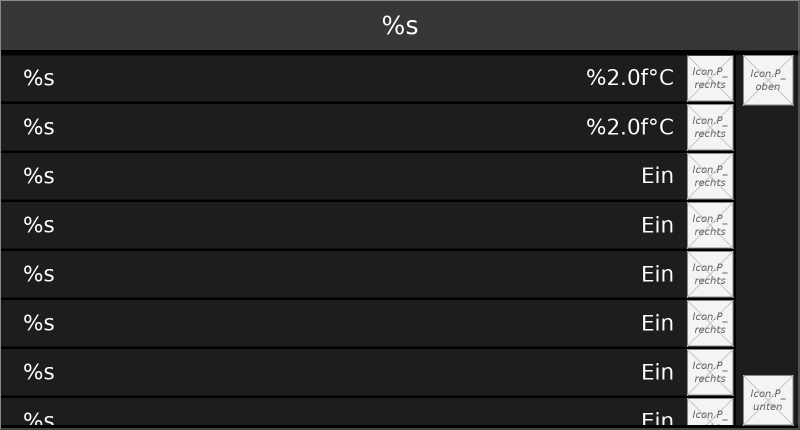
VISUALIZATION SW_WG_UWP_Verd_Liste  // 800x430
VAR_IN_OUT
	FB_GR2:GR_2;
END_VAR

VAR_INPUT
	i_Titel:INT;
END_VAR

VAR
	i_verschieben:INT;
 END_VAR
    Rectangle (0,55 733x46)
    Label (20,55 479x46), "%s"
    Rectangle (0,104 733x46)
    Label (20,104 479x46), "%s"
    Rectangle (547,55 130x45), "%2.0f°C", text variable: FB_GR2.f_AT
    Rectangle (547,104 130x46), "%2.0f°C", text variable: FB_GR2.f_RefPunkt_TO1
    Image (687,55 46x46), image: Icon.P_rechts
        OnMouseClick: execute { GWP_Library.Visu.i_Frame_Index:=1; }
    Image (687,104 46x46), image: Icon.P_rechts
    Rectangle (0,153 733x46)
    Label (20,153 479x46), "%s"
    Rectangle (0,202 733x46)
    Label (20,202 479x46), "%s"
    Rectangle (0,251 733x46)
    Label (20,251 479x46), "%s"
    Rectangle (0,300 733x46)
    Label (20,300 479x46), "%s"
    Rectangle (0,349 733x46)
    Label (20,349 479x46), "%s"
    Rectangle (0,398 733x46)
    Label (20,398 479x46), "%s"
    Rectangle (0,447 733x46)
    Label (20,447 479x46), "%s"
    Rectangle (0,496 733x46)
    Label (20,496 479x46), "%s"
    Rectangle (0,545 733x46)
    Label (20,545 479x46), "%s"
    Rectangle (547,153 130x45), "Ein"
    Rectangle (547,202 130x46), "Ein"
    Rectangle (547,251 130x46), "Ein"
    Rectangle (547,300 130x46), "Ein"
    Rectangle (547,349 130x46), "Ein"
    Rectangle (547,447 130x46), "Ein"
    Rectangle (547,398 130x46), "Ein"
    Rectangle (547,496 130x46), "Ein"
    Rectangle (547,545 130x46), "Ein"
    Image (687,153 46x46), image: Icon.P_rechts
        OnMouseClick: execute { GWP_Library.Visu.i_Frame_Index:=3; }
    Image (687,545 46x46), image: Icon.P_rechts
    Image (687,496 46x46), image: Icon.P_rechts
    Image (687,447 46x46), image: Icon.P_rechts
    Image (687,398 46x46), image: Icon.P_rechts
    Image (687,349 46x46), image: Icon.P_rechts
    Image (687,300 46x46), image: Icon.P_rechts
    Image (687,251 46x46), image: Icon.P_rechts
    Image (687,202 46x46), image: Icon.P_rechts
    Rectangle (0,594 733x46)
    Label (20,594 479x46), "%s"
    Rectangle (547,594 130x45), "Ein"
    Image (687,594 46x46), image: Icon.P_rechts
    Image (79,430 50x50), image: Icon.zurueck
        OnMouseClick:  Assign=Sollwertmenu_Waermegewinnung, Type=Assignment
        OnMouseClick: execute { i_verschieben:=0; }
    Rectangle (0,0 800x50), "%s", text list: 'Sprachen', text index: i_Titel
    Group (736,55 64x370)
        Rectangle (0,0 64x370)
        Image (7,320 50x50), image: Icon.P_unten
            OnMouseClick: execute {
                IF i_verschieben<0 THEN
                	i_verschieben:=i_verschieben+53;
                End_if
            }
        Image (7,0 50x50), image: Icon.P_oben
            OnMouseClick: execute {
                IF  i_verschieben>-200 THEN
                	i_verschieben:=i_verschieben-53;
                End_if
            }
    Rectangle (0,50 733x5)
    Rectangle (0,425 733x5)
END_VISUALIZATION

// VISUs/Sollwertmenu_9/Wärmegewinnung/Sollwertmenu_Waermegewinnung
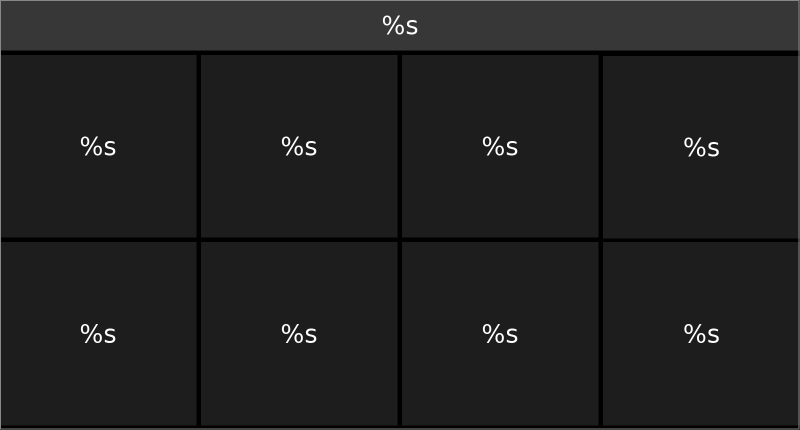
VISUALIZATION Sollwertmenu_Waermegewinnung  // 800x430
    Rectangle (0,0 800x50), "%s", text list: 'Sprachen', text index: 4
    Rectangle (0,55 196x182), "%s", text list: 'Sprachen', text index: 5
        OnMouseClick:  Assign=SW_WG_UWP_Verd, Type=Assignment
    Rectangle (201,55 196x182), "%s", text list: 'Sprachen', text index: 6
        OnMouseClick:  Assign=IO_Auswahl, Type=Assignment
    Rectangle (402,55 196x182), "%s", text list: 'Sprachen', text index: 7
    Rectangle (603,56 197x182), "%s", text list: 'Sprachen', text index: 8
    Rectangle (0,242 196x183), "%s", text list: 'Sprachen', text index: 9
    Rectangle (201,242 196x183), "%s", text list: 'Sprachen', text index: 10
    Rectangle (402,242 196x183), "%s", text list: 'Sprachen', text index: 11
    Rectangle (603,242 197x183), "%s", text list: 'Sprachen', text index: 12
    Image (125,430 50x50), image: Icon.zurueck
        OnMouseClick:  Assign=Sollwertmenu, Type=Assignment
    Frame (0,430 800x50)
        shows Fusszeile_50()
END_VISUALIZATION

// VISUs/Sollwertmenu_9/_SW_Heizgruppe
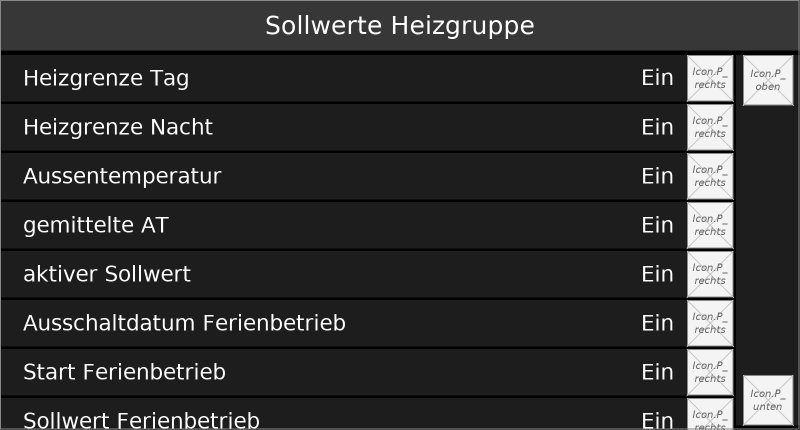
VISUALIZATION _SW_Heizgruppe  // 800x430
    Rectangle (0,0 800x50), "Sollwerte Heizgruppe"
    Rectangle (0,55 733x46)
    Label (20,55 479x46), "Heizgrenze Tag"
    Rectangle (0,104 733x46)
    Label (20,104 479x46), "Heizgrenze Nacht"
    Rectangle (0,153 733x46)
    Label (20,153 479x46), "Aussentemperatur"
    Rectangle (0,202 733x46)
    Label (20,202 479x46), "gemittelte AT"
    Rectangle (0,251 733x46)
    Label (20,251 479x46), "aktiver Sollwert"
    Rectangle (0,300 733x46)
    Label (20,300 479x46), "Ausschaltdatum Ferienbetrieb"
    Rectangle (0,349 733x46)
    Label (20,349 479x46), "Start Ferienbetrieb"
    Rectangle (547,55 130x45), "Ein"
    Rectangle (547,104 130x46), "Ein"
    Rectangle (547,153 130x46), "Ein"
    Rectangle (547,202 130x46), "Ein"
    Rectangle (547,251 130x46), "Ein"
    Rectangle (547,349 130x46), "Ein"
    Rectangle (547,300 130x46), "Ein"
    Image (687,55 46x46), image: Icon.P_rechts
    Rectangle (0,398 733x46)
    Label (20,398 479x46), "Sollwert Ferienbetrieb"
    Rectangle (547,398 130x46), "Ein"
    Image (687,398 46x46), image: Icon.P_rechts
    Image (687,349 46x46), image: Icon.P_rechts
    Image (687,300 46x46), image: Icon.P_rechts
    Image (687,251 46x46), image: Icon.P_rechts
    Image (687,202 46x46), image: Icon.P_rechts
    Image (687,153 46x46), image: Icon.P_rechts
    Image (687,104 46x46), image: Icon.P_rechts
    Rectangle (736,55 64x370)
    Image (743,55 50x50), image: Icon.P_oben
        OnMouseClick: write the text variable via Default
    Image (743,375 50x50), image: Icon.P_unten
    Rectangle (0,447 733x46)
    Label (20,447 479x46), "Restzeit Ferienbetrieb"
    Rectangle (547,447 130x46), "Ein"
    Image (687,447 46x46), image: Icon.P_rechts
END_VISUALIZATION

// VISUs/Sollwertmenu_9/_SW_Speicher_BWW
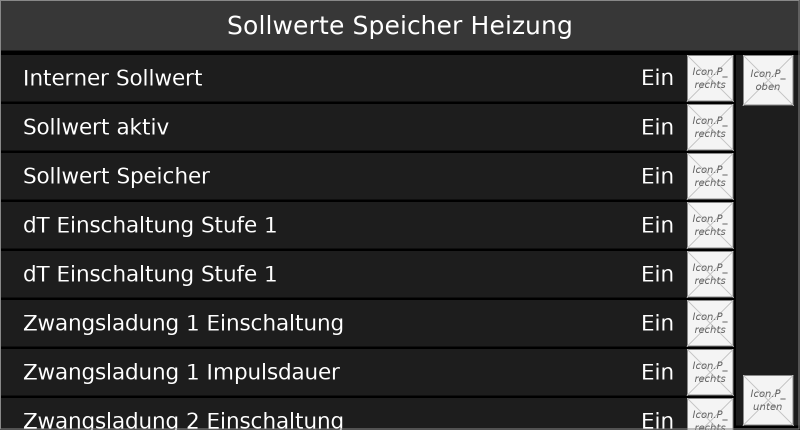
VISUALIZATION _SW_Speicher_BWW  // 800x430
VAR_IN_OUT
	auf:BOOL;
	
END_VAR
    Rectangle (0,0 800x50), "Sollwerte Speicher Heizung"
    Rectangle (0,55 733x46)
    Label (20,55 479x46), "Interner Sollwert"
    Rectangle (0,104 733x46)
    Label (20,104 479x46), "Sollwert aktiv"
    Rectangle (0,153 733x46)
    Label (20,153 479x46), "Sollwert Speicher"
    Rectangle (0,202 733x46)
    Label (20,202 479x46), "dT Einschaltung Stufe 1"
    Rectangle (0,251 733x46)
    Label (20,251 479x46), "dT Einschaltung Stufe 1"
    Rectangle (0,300 733x46)
    Label (20,300 479x46), "Zwangsladung 1 Einschaltung"
    Rectangle (0,349 733x46)
    Label (20,349 479x46), "Zwangsladung 1 Impulsdauer"
    Rectangle (547,55 130x45), "Ein"
    Rectangle (547,104 130x46), "Ein"
    Rectangle (547,153 130x46), "Ein"
    Rectangle (547,202 130x46), "Ein"
    Rectangle (547,251 130x46), "Ein"
    Rectangle (547,349 130x46), "Ein"
    Rectangle (547,300 130x46), "Ein"
    Image (687,55 46x46), image: Icon.P_rechts
    Rectangle (0,398 733x46)
    Label (20,398 479x46), "Zwangsladung 2 Einschaltung"
    Rectangle (547,398 130x46), "Ein"
    Image (687,398 46x46), image: Icon.P_rechts
    Image (687,349 46x46), image: Icon.P_rechts
    Image (687,300 46x46), image: Icon.P_rechts
    Image (687,251 46x46), image: Icon.P_rechts
    Image (687,202 46x46), image: Icon.P_rechts
    Image (687,153 46x46), image: Icon.P_rechts
    Image (687,104 46x46), image: Icon.P_rechts
    Rectangle (736,55 64x370)
    Image (743,55 50x50), image: Icon.P_oben
        OnMouseClick: write the text variable via Default
    Image (743,375 50x50), image: Icon.P_unten
    Rectangle (0,447 733x46)
    Label (20,447 479x46), "Zwangsladung 2 Impulsdauer"
    Rectangle (547,447 130x46), "Ein"
    Image (687,447 46x46), image: Icon.P_rechts
END_VISUALIZATION

// VISUs/Sollwertmenu_9/_SW_Speicher_Heizung_1
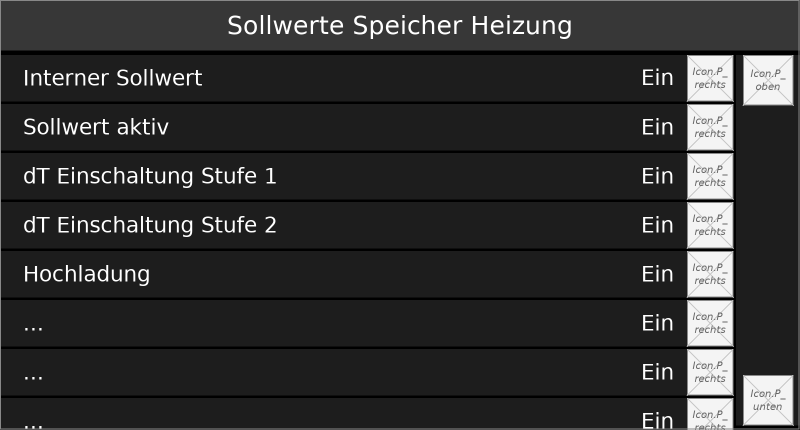
VISUALIZATION _SW_Speicher_Heizung_1  // 800x430
VAR_IN_OUT
	auf:BOOL;
	
END_VAR
    Rectangle (0,0 800x50), "Sollwerte Speicher Heizung"
    Rectangle (0,55 733x46)
    Label (20,55 479x46), "Interner Sollwert"
    Rectangle (0,104 733x46)
    Label (20,104 479x46), "Sollwert aktiv"
    Rectangle (0,153 733x46)
    Label (20,153 479x46), "dT Einschaltung Stufe 1"
    Rectangle (0,202 733x46)
    Label (20,202 479x46), "dT Einschaltung Stufe 2"
    Rectangle (0,251 733x46)
    Label (20,251 479x46), "Hochladung"
    Rectangle (0,300 733x46)
    Label (20,300 479x46), "..."
    Rectangle (0,349 733x46)
    Label (20,349 479x46), "..."
    Rectangle (0,398 733x46)
    Label (20,398 479x46), "..."
    Rectangle (547,55 130x45), "Ein"
    Rectangle (547,104 130x46), "Ein"
    Rectangle (547,153 130x46), "Ein"
    Rectangle (547,202 130x46), "Ein"
    Rectangle (547,251 130x46), "Ein"
    Rectangle (547,349 130x46), "Ein"
    Rectangle (547,300 130x46), "Ein"
    Rectangle (547,398 130x46), "Ein"
    Image (687,55 46x46), image: Icon.P_rechts
    Image (687,398 46x46), image: Icon.P_rechts
    Image (687,349 46x46), image: Icon.P_rechts
    Image (687,300 46x46), image: Icon.P_rechts
    Image (687,251 46x46), image: Icon.P_rechts
    Image (687,202 46x46), image: Icon.P_rechts
    Image (687,153 46x46), image: Icon.P_rechts
    Image (687,104 46x46), image: Icon.P_rechts
    Group (736,55 64x370)
        Rectangle (0,0 64x370)
        Image (7,0 50x50), image: Icon.P_oben
            OnMouseClick: write the text variable via Default
        Image (7,320 50x50), image: Icon.P_unten
END_VISUALIZATION

// VISUs/Sollwertmenu_9/_SW_Speicher_Kaltwasser
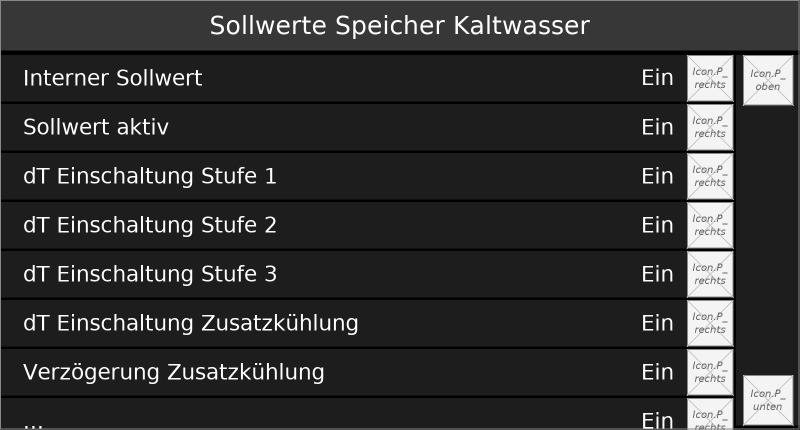
VISUALIZATION _SW_Speicher_Kaltwasser  // 800x430
    Rectangle (0,0 800x50), "Sollwerte Speicher Kaltwasser"
    Rectangle (0,55 733x46)
    Label (20,55 479x46), "Interner Sollwert"
    Rectangle (0,104 733x46)
    Label (20,104 479x46), "Sollwert aktiv"
    Rectangle (0,153 733x46)
    Label (20,153 479x46), "dT Einschaltung Stufe 1"
    Rectangle (0,202 733x46)
    Label (20,202 479x46), "dT Einschaltung Stufe 2"
    Rectangle (0,251 733x46)
    Label (20,251 479x46), "dT Einschaltung Stufe 3"
    Rectangle (0,300 733x46)
    Label (20,300 479x46), "dT Einschaltung Zusatzkühlung"
    Rectangle (0,349 733x46)
    Label (20,349 479x46), "Verzögerung Zusatzkühlung"
    Rectangle (0,398 733x46)
    Label (20,398 479x46), "..."
    Rectangle (0,447 733x46)
    Label (20,447 479x46), "..."
    Rectangle (0,496 733x46)
    Label (20,496 479x46), "..."
    Group (736,55 64x370)
        Rectangle (0,0 64x370)
        Image (7,0 50x50), image: Icon.P_oben
            OnMouseClick: write the text variable via Default
        Image (7,320 50x50), image: Icon.P_unten
    Rectangle (547,55 130x45), "Ein"
    Rectangle (547,104 130x46), "Ein"
    Rectangle (547,153 130x46), "Ein"
    Rectangle (547,202 130x46), "Ein"
    Rectangle (547,251 130x46), "Ein"
    Rectangle (547,349 130x46), "Ein"
    Rectangle (547,300 130x46), "Ein"
    Rectangle (547,398 130x46), "Ein"
    Rectangle (547,496 130x46), "Ein"
    Rectangle (547,447 130x46), "Ein"
    Image (687,55 46x46), image: Icon.P_rechts
    Image (687,447 46x46), image: Icon.P_rechts
    Image (687,398 46x46), image: Icon.P_rechts
    Image (687,349 46x46), image: Icon.P_rechts
    Image (687,300 46x46), image: Icon.P_rechts
    Image (687,251 46x46), image: Icon.P_rechts
    Image (687,202 46x46), image: Icon.P_rechts
    Image (687,153 46x46), image: Icon.P_rechts
    Image (687,104 46x46), image: Icon.P_rechts
    Image (687,496 46x46), image: Icon.P_rechts
END_VISUALIZATION

// VISUs/Sollwertmenu_9/_SW_Waermegewinnung
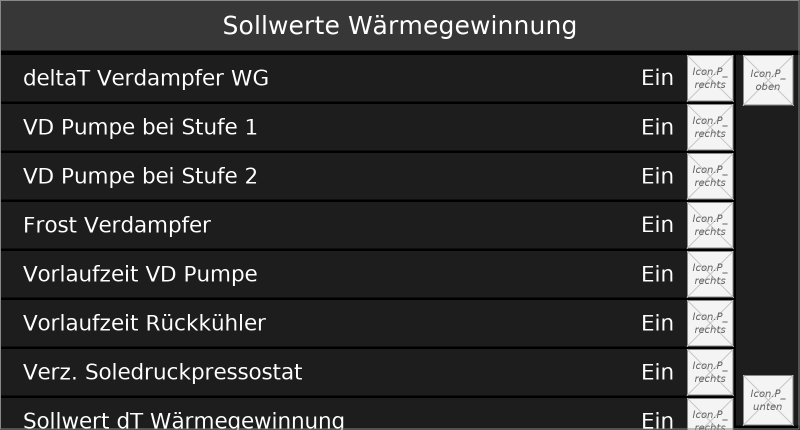
VISUALIZATION _SW_Waermegewinnung  // 800x430
    Rectangle (0,0 800x50), "Sollwerte Wärmegewinnung"
    Rectangle (0,55 733x46)
    Label (20,55 479x46), "deltaT Verdampfer WG"
    Rectangle (0,104 733x46)
    Label (20,104 479x46), "VD Pumpe bei Stufe 1"
    Rectangle (0,153 733x46)
    Label (20,153 479x46), "VD Pumpe bei Stufe 2"
    Rectangle (547,55 130x45), "Ein"
    Rectangle (547,104 130x46), "Ein"
    Rectangle (547,153 130x46), "Ein"
    Image (687,55 46x46), image: Icon.P_rechts
    Image (687,153 46x46), image: Icon.P_rechts
    Image (687,104 46x46), image: Icon.P_rechts
    Group (736,55 64x370)
        Rectangle (0,0 64x370)
        Image (7,0 50x50), image: Icon.P_oben
            OnMouseClick: write the text variable via Default
        Image (7,320 50x50), image: Icon.P_unten
    Rectangle (0,202 733x46)
    Label (20,202 479x46), "Frost Verdampfer"
    Rectangle (0,251 733x46)
    Label (20,251 479x46), "Vorlaufzeit VD Pumpe"
    Rectangle (0,300 733x46)
    Label (20,300 479x46), "Vorlaufzeit Rückkühler"
    Rectangle (0,349 733x46)
    Label (20,349 479x46), "Verz. Soledruckpressostat"
    Rectangle (0,398 733x46)
    Label (20,398 479x46), "Sollwert dT Wärmegewinnung"
    Rectangle (0,447 733x46)
    Label (20,447 479x46), "Sollwert Temp. Austritt"
    Rectangle (0,496 733x46)
    Label (20,496 479x46), "..."
    Rectangle (0,545 733x46)
    Label (20,545 479x46), "..."
    Rectangle (547,202 130x45), "Ein"
    Rectangle (547,251 130x46), "Ein"
    Rectangle (547,300 130x46), "Ein"
    Rectangle (547,349 130x46), "Ein"
    Rectangle (547,398 130x46), "Ein"
    Rectangle (547,496 130x46), "Ein"
    Rectangle (547,447 130x46), "Ein"
    Rectangle (547,545 130x46), "Ein"
    Image (687,202 46x46), image: Icon.P_rechts
    Image (687,545 46x46), image: Icon.P_rechts
    Image (687,496 46x46), image: Icon.P_rechts
    Image (687,447 46x46), image: Icon.P_rechts
    Image (687,398 46x46), image: Icon.P_rechts
    Image (687,349 46x46), image: Icon.P_rechts
    Image (687,300 46x46), image: Icon.P_rechts
    Image (687,251 46x46), image: Icon.P_rechts
END_VISUALIZATION

// VISUs/Sollwertmenu_9/Sollwertmenu_Waermesenke
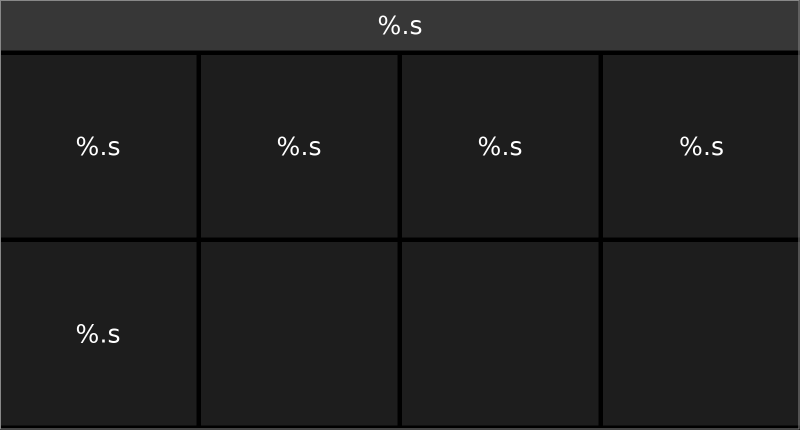
VISUALIZATION Sollwertmenu_Waermesenke  // 800x430
    Rectangle (0,0 800x50), "%.s"
    Rectangle (0,55 196x182), "%.s"
    Rectangle (201,55 196x182), "%.s"
    Rectangle (402,55 196x182), "%.s"
    Rectangle (603,55 197x182), "%.s"
    Rectangle (0,242 196x183), "%.s"
    Rectangle (201,242 196x183)
    Rectangle (402,242 196x183)
    Rectangle (603,242 197x183)
    Frame (0,430 800x50)
        shows Fusszeile_50()
    Image (125,430 50x50), image: Icon.zurueck
        OnMouseClick:  Assign=Sollwertmenu, Type=Assignment
END_VISUALIZATION

// VISUs/Sollwertmenu_9/SW_Waermepumpe
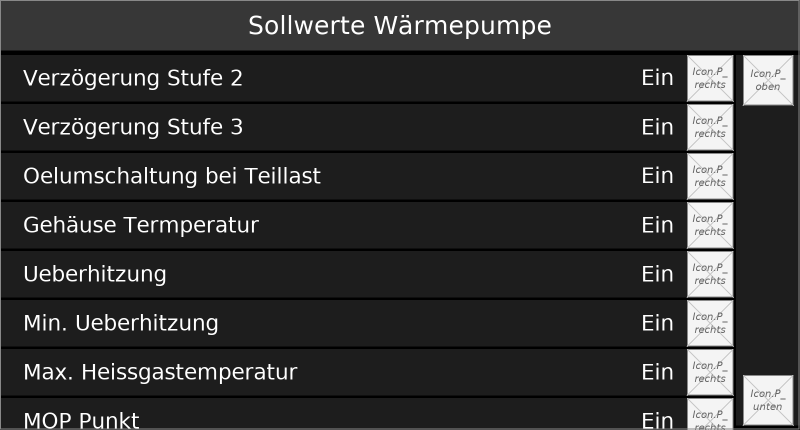
VISUALIZATION SW_Waermepumpe  // 800x430
VAR_IN_OUT
	
END_VAR

VAR_INPUT
	i_Titel:INT;
END_VAR

 VAR
	auf:BOOL:=0;
	ab:BOOL:=0;
	verschieben:INT:=0;
 END_VAR
    Rectangle (736,55 64x370)
    Image (743,55 50x50), text list: '', image: Icon.P_oben
        OnMouseClick:  ToggleVariable=auf
        OnMouseClick: execute {
            IF auf THEN
            	verschieben:=verschieben-50;
            	auf:=0;
            END_IF
        }
    Image (743,375 50x50), image: Icon.P_unten
        OnMouseClick:  ToggleVariable=ab
        OnMouseClick: execute {
            IF ab THEN
            	verschieben:=verschieben+50;
            	ab:=0;
            END_IF
        }
    Group (0,55 733x1026)
        Rectangle (0,0 733x46)
        Label (20,0 479x46), "Verzögerung Stufe 2"
        Rectangle (0,49 733x46)
        Label (20,49 479x46), "Verzögerung Stufe 3"
        Rectangle (547,0 130x45), "Ein"
        Rectangle (547,49 130x46), "Ein"
        Image (687,0 46x46), image: Icon.P_rechts
            OnMouseClick: FrameSelectionChange Selection=Selection=-1, GlobSel=IndExpr=2, AssignDir=Test_SW_WP.GenElemInst_5, AssignType=Directly, SelType=Globally
        Image (687,49 46x46), image: Icon.P_rechts
        Rectangle (0,98 733x46)
        Label (20,98 479x46), "Oelumschaltung bei Teillast"
        Rectangle (0,147 733x46)
        Label (20,147 479x46), "Gehäuse Termperatur"
        Rectangle (0,196 733x46)
        Label (20,196 479x46), "Ueberhitzung"
        Rectangle (0,245 733x46)
        Label (20,245 479x46), "Min. Ueberhitzung"
        Rectangle (0,294 733x46)
        Label (20,294 479x46), "Max. Heissgastemperatur"
        Rectangle (0,343 733x46)
        Label (20,343 479x46), "MOP Punkt"
        Rectangle (0,392 733x46)
        Label (20,392 479x46), "Verzögerung Alarm EEV"
        Rectangle (0,441 733x46)
        Label (20,441 479x46), "deltaP Oeldruck"
        Rectangle (0,490 733x46)
        Label (20,490 479x46), "Verzögerung Alarm Oeldruck"
        Rectangle (547,98 130x45), "Ein"
        Rectangle (547,147 130x46), "Ein"
        Rectangle (547,196 130x46), "Ein"
        Rectangle (547,245 130x46), "Ein"
        Rectangle (547,294 130x46), "Ein"
        Rectangle (547,392 130x46), "Ein"
        Rectangle (547,343 130x46), "Ein"
        Rectangle (547,441 130x46), "Ein"
        Rectangle (547,490 130x46), "Ein"
        Image (687,98 46x46), image: Icon.P_rechts
            OnMouseClick: execute { GWP_Library.Visu.i_Frame_Index:=3; }
        Image (687,490 46x46), image: Icon.P_rechts
        Image (687,441 46x46), image: Icon.P_rechts
        Image (687,392 46x46), image: Icon.P_rechts
        Image (687,343 46x46), image: Icon.P_rechts
        Image (687,294 46x46), image: Icon.P_rechts
        Image (687,245 46x46), image: Icon.P_rechts
        Image (687,196 46x46), image: Icon.P_rechts
        Image (687,147 46x46), image: Icon.P_rechts
        Rectangle (0,539 733x46)
        Label (20,539 479x46), "Niederdruckalarm"
        Rectangle (0,588 733x46)
        Label (20,588 479x46), "Verzögerung Niederdruck"
        Rectangle (0,637 733x46)
        Label (20,637 479x46), "Verzögerung Niederdruck anf."
        Rectangle (0,686 733x46)
        Label (20,686 479x46), "Hochdruckalarm"
        Rectangle (0,735 733x46)
        Label (20,735 479x46), "Verzögerung Hochdruck"
        Rectangle (0,784 733x46)
        Label (20,784 479x46), "Anzahl ND bis Auslösung AL"
        Rectangle (0,833 733x46)
        Label (20,833 479x46), "Anzahl HD bis Auslösung AL"
        Rectangle (0,882 733x46)
        Label (20,882 479x46), "Sperrzeit WP nach ND/HD"
        Rectangle (0,931 733x46)
        Label (20,931 479x46), "Tage Reset Zähler ND/HD"
        Rectangle (0,980 733x46)
        Label (20,980 479x46), "..."
        Rectangle (547,539 130x45), "Ein"
        Rectangle (547,588 130x46), "Ein"
        Rectangle (547,637 130x46), "Ein"
        Rectangle (547,686 130x46), "Ein"
        Rectangle (547,735 130x46), "Ein"
        Rectangle (547,833 130x46), "Ein"
        Rectangle (547,784 130x46), "Ein"
        Rectangle (547,882 130x46), "Ein"
        Rectangle (547,980 130x46), "Ein"
        Rectangle (547,931 130x46), "Ein"
        Image (687,539 46x46), image: Icon.P_rechts
        Image (687,931 46x46), image: Icon.P_rechts
        Image (687,882 46x46), image: Icon.P_rechts
        Image (687,833 46x46), image: Icon.P_rechts
        Image (687,784 46x46), image: Icon.P_rechts
        Image (687,735 46x46), image: Icon.P_rechts
        Image (687,686 46x46), image: Icon.P_rechts
        Image (687,637 46x46), image: Icon.P_rechts
        Image (687,588 46x46), image: Icon.P_rechts
        Image (687,980 46x46), image: Icon.P_rechts
    Rectangle (0,0 800x50), "Sollwerte Wärmepumpe", text list: 'Sprachen', text index: i_Titel
    Rectangle (883,211 150x30)
        OnMouseClick:  Assign=SW_Einst_WP_Verz_Stufe2, Type=Assignment
END_VISUALIZATION

// VISUs/Zeitprogramm/Wochenuhr_W7
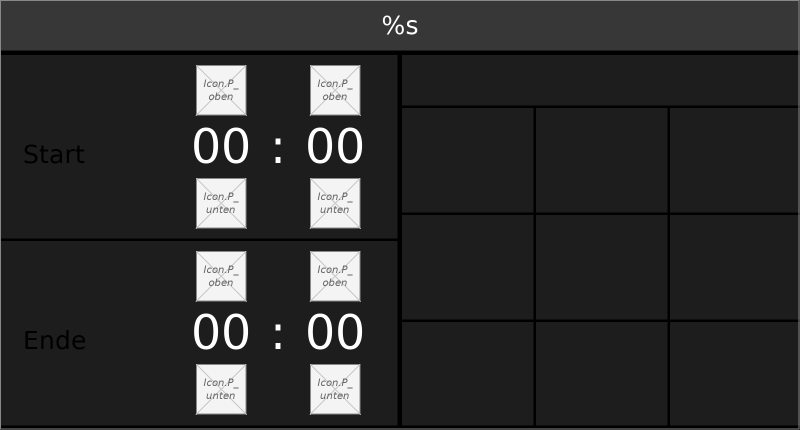
VISUALIZATION Wochenuhr_W7  // 800x430
    Rectangle (0,0 800x50), "%s", text list: 'Sprachen', text index: 52
    Rectangle (402,55 398x50)
    Rectangle (402,108 131x104)
    Rectangle (536,108 131x104)
    Rectangle (670,108 130x104)
    Rectangle (402,215 131x104)
    Rectangle (536,215 131x104)
    Rectangle (670,215 130x104)
    Rectangle (402,322 131x103)
    Rectangle (536,322 131x103)
    Rectangle (670,322 130x103)
    Group (0,55 397x183)
        Rectangle (0,0 397x183)
        Rectangle (263,49 30x84), ":"
        Rectangle (179,49 84x84), "00"
        Rectangle (293,49 84x84), "00"
        Rectangle (20,57 150x84), "Start"
        Image (196,10 50x50), image: Icon.P_oben
        Image (196,123 50x50), image: Icon.P_unten
        Image (310,10 50x50), image: Icon.P_oben
        Image (310,123 50x50), image: Icon.P_unten
    Rectangle (0,241 397x184)
    Rectangle (263,290 30x84), ":"
    Rectangle (179,290 84x84), "00"
    Rectangle (293,290 84x84), "00"
    Rectangle (20,298 150x84), "Ende"
    Image (196,251 50x50), image: Icon.P_oben
    Image (196,364 50x50), image: Icon.P_unten
    Image (310,251 50x50), image: Icon.P_oben
    Image (310,364 50x50), image: Icon.P_unten
END_VISUALIZATION

// VISUs/test_1
VISUALIZATION test_1  // 800x400
END_VISUALIZATION

(* text list Sprachen (id | default | Deutsch | Englisch | De)
  100 | Verzoegerung Stufe 2 |  |  | 
  101 | Verzögerung Stufe 1 |  |  | 
  0 | Wärmegewinnung |  |  | 
  1 | Wärmepumpe |  |  | 
  2 | Waermesenke |  |  | 
  3 | Sollwertmenue |  |  | 
  4 | Sollwerte Waermegewinnung |  |  | 
  5 | UWP Verd. |  |  | 
  6 | Erdsonde |  |  | 
  7 | Grundwasser |  |  | 
  8 | Luft |  |  | 
  9 | Tiefhaltung |  |  | 
  10 | Abtauspeicher |  |  | 
  11 | Abtauungen |  |  | 
  12 | Abwaerme |  |  | 
  13 |  |  |  | 
  14 | Sollwerte Waermepumpe |  |  | 
  15 | EEV |  |  | 
  16 | Einsatzgrenzen |  |  | 
  17 | Verdichter |  |  | 
  18 | Allgemein |  |  | 
  19 | Sollwerte Wärmesenke |  |  | 
  20 | UWP Verflüssiger |  |  | 
  21 | HWP |  |  | 
  22 | TWW |  |  | 
  23 | Heizgruppe |  |  | 
  24 | Hochhaltung |  |  | 
  25 | Sollwerte UWP Verdampfer |  |  | 
  26 | Sollwerte Erdsonden |  |  | 
  27 | Sollwerte Luft |  |  | 
  28 | Sollwerte Abwärme |  |  | 
  29 | Sollwerte Tiefhaltung |  |  | 
  30 | Sollwertänderung Zeit |  |  | 
  31 | Infoseite |  |  | 
  32 | Hauptmenue |  |  | 
  33 | Sprachen |  |  | 
  34 | Login |  |  | 
  35 | Sollwerte |  |  | 
  36 | Verlaufsdiagramm |  |  | 
  37 | Uhrzeit einstellen |  |  | 
  38 | IBN |  |  | 
  39 | Konfiguration |  |  | 
  40 | Kontakt |  |  | 
  41 | Ein/Aus Waermepumpe |  |  | 
  42 | Ein |  |  | 
  43 | Aus |  |  | 
  44 | IO-Auswahl |  |  | 
  45 | Digitale Eingaenge |  |  | 
  46 | Digitale Ausgaenge |  |  | 
  47 | Analoge Eingaenge |  |  | 
  48 | Analoge Ausgaenge |  |  | 
  49 | Status |  |  | 
  50 | Offset |  |  | 
  51 | Istwert |  |  | 
  52 | Wochenschaltuhr |  |  | 
  54 |  |  |  | 
   |  |  |  |  *)
